Yaskawa INFORM job: M004GUID.JBI

/JOB
//NAME M004GUID
//POS
///NPOS 0,0,0,0,0,0
//INST
///DATE 2019/08/05 22:05
///ATTR SC,RW,MC
///GROUP1 RB1
///LVARS 0,0,3,0,0,0,0,0
NOP
GETARG LD000 IARG#(1)
SET D070 LD000
SET B069 0
SKILLSND "Comm004Guide"
WAIT B069=1
END
